PROGRAM MAIN
VAR
	fbPowerShell:FB_PowerShell; 
	xRunSample1:BOOL;
	xRunSample2: BOOL;
	xRunSample3: BOOL;
	xToggleValue:BOOL;
END_VAR

//This must be called every PLC scan. 
fbPowerShell(udiErrId=> , xBusy=> , xError=> );

IF xRunSample1 THEN //Start HERE!!!
	xRunSample1:=FALSE;
	fbPowerShell.PowerShellLine:='Write-Output  "Hello World!!!"';
	fbPowerShell.PowerShellLine:='Read-Host -Prompt "Press Enter to exit"';
END_IF


IF xRunSample2 THEN //Example varient swap. Copys a new PLC program into boot folder so the PLC project can change. Warning, does reboot PC.
	xRunSample2:=FALSE;
	fbPowerShell.PowerShellLine:='Remove-Item -path C:\TwinCAT\3.1\Boot\* -Exclude *.db -recurse';
	fbPowerShell.PowerShellLine:='Copy-Item -Path "C:\Varients\VarientA\*" -Destination C:\TwinCAT\3.1\Boot -Recurse';
	fbPowerShell.PowerShellLine:='Restart-Computer'; 
END_IF


IF xRunSample3 THEN //Example to read or write to a PLC tag from powershell. If you need feedback from your Powershell code this is how you do it.
	xRunSample3:=FALSE;
	//Option #1. I personally prefer this because it requires no special setup. However, the code must be successful at finding the TwinCAT.Ads.dll. 
	fbPowerShell.PowerShellLine:='$$Path = Get-Childitem –Path "C:\TwinCAT\AdsApi\.NET\" -Recurse -Include "TwinCAT.Ads.dll" | Where-Object {-not $$_.DirectoryName.Contains("CE")}  | Select-Object -First 1';  //This is designed to find the ADS library for you. It may fail
	fbPowerShell.PowerShellLine:='Add-Type -Path $$Path';  //UPDATE the Path here to were your ADS.net library files are. Just change $$Path to "full Path to TwinCAT.Ads.dll" 	
	fbPowerShell.PowerShellLine:='$$tcClient = New-Object TwinCAT.Ads.TcAdsClient'; //Create TwinCAT client
	fbPowerShell.PowerShellLine:='$$tcClient.Connect(851)'; //Connect to PLC
	fbPowerShell.PowerShellLine:='$$value = $$tcClient.ReadSymbol("Main.xToggleValue", "Boolean","")';	//Read a tag and write it to "value"
	fbPowerShell.PowerShellLine:='$$tcClient.WriteSymbol("Main.xToggleValue", -not $$value , 0)';	//write a tag by toggling it
	fbPowerShell.PowerShellLine:='$$tcClient.Disconnect()';	 //Disconnect
	
	
	//Option #2. Some beleive this to be the correct way but requires installing a module and setting an environment path in windows.
	//Warning, requires TE1000 TwinCAT 3 | ADS Powershell module installed. Requires running special powershell commands to install.
	(*
	fbPowerShell.PowerShellLine:='$$session = New-TcSession -Port 851';
	fbPowerShell.PowerShellLine:='$$symbol = $$session | get-TcSymbol -Path $'Main.xToggleValue$'';
	//fbPowerShell.PowerShellLine:='$$symbol | Read-TcValue';
	fbPowerShell.PowerShellLine:='$$symbol | Write-TcValue -Value 1 -force -Quiet';
	*)
END_IF



(*
For special characters. 
$$ = $    
$' = '    
$r = carriage return
https://infosys.beckhoff.com/english.php?content=../content/1033/tc3_plc_intro/2529327243.html&id=


Helpful power shell code samples.
To pause the powersshell to read the output values.  Read-Host -Prompt "Press Enter to exit"

Get-NetIPAddress -AddressFamily IPv4
New-NetIPAddress -InterfaceIndex 12 -IPAddress 192.168.0.1

*)

END_PROGRAM

(* stored: Version 1.1.0.1, ProductVersion 3.1.4024.12
   POU MAIN: Id {bb0bb8c9-51d4-4604-868f-f5d016f9a231}, SpecialFunc None *)
